// TIA Portal V17 export
// export: Created 2024-08-09T12:53:13.545274Z, ExportSetting WithDefaults, DisplayName Totally Integrated Automation Portal, DisplayVersion V17 Update 7, DisplayName TIA Portal Openness, DisplayVersion V17 Update 7, DisplayName TIA Portal Version Control Interface, DisplayVersion V17, DisplayName STEP 7 Professional, DisplayVersion V17 Update 7, DisplayName STEP 7 Safety, DisplayVersion V17 Update 6, DisplayName WinCC Professional, DisplayVersion V17 Update 7
VAR_GLOBAL   // PLC tag table "Transfert"
END_VAR
VAR_GLOBAL CONSTANT   // user constants
   NIV_CIRTRANS_DEBUT_LOT : USInt := 1;
   NIV_CIRTRANS_CIR_TRANS_PRET : USInt := 50;
   NIV_CIRTRANS_CIR_FIN_LOT : USInt := 255;
END_VAR
